INTERFACE ITF_Can_Supply EXTENDS ITF_PackML

END_INTERFACE

(* stored: Version 1.1.0.1, ProductVersion 3.1.4024.12
   Itf ITF_Can_Supply: Id {be7d18ee-7936-4035-920e-6c9d83390de9} *)
